Yaskawa INFORM job: SET_UFRAME.JBI

/JOB
//NAME SET_UFRAME
///FOLDERNAME TWINCAT_KOMMUNIKATION
//POS
///NPOS 0,0,0,0,0,0
//ALIAS
///LVARS 0,1,0,0,0,0,0,0
LI000 UFRAME_NR
//ARGINFO
///ARGTYPE I,,,,,,,
///COMMENT
UFRAME_NR







//INST
///DATE 2021/04/27 10:40
///ATTR SC,RW
///LVARS 0,1,0,0,0,0,0,0
NOP
GETARG UFRAME_NR IARG#(1)
SETREG MREG#(68) UFRAME_NR
END
